FUNCTION_BLOCK IA_COGSOGRapidUpdate (* ISOBUS Adapter for Course Over Ground and Speed Over Ground (Rapid Update) *)
  (* Standard: NMEA 2000; Classification: PGN 129026; Description: Copyright (c) 2024-2026 HR Agrartechnik GmbH This program and the accompanying materials are made available under the terms of the Eclipse Public License 2.0 which is available at https://www.eclipse.org/legal/epl-2.0/ SPDX-License-Identifier: EPL-2.0 *)
  (* Version 1.4, 2026-09-17, Franz Höpfinger, HR Agrartechnik GmbH, Dokumentation (Franz: 'das passt, wir dokumentieren das in den Bausteinen. E_D_FF ist ein IEC 61499 Standardbaustein, wir halten uns STRENG an die Norm. E_D_FF_ANY ist davon abgeleitet, sollte sich gleich verhalten'): E_D_FF_Timeout (E_D_FF, IEC 61499-1 Annex A Standardbaustein) feuert EO NICHT beim allerersten CLK, wenn der erste echte Wert mit dem default-initialisierten Vergleichszustand (FALSE) uebereinstimmt - bleibt I_CORE.Q_timeout von Anfang an FALSE (Normalfall, kein Timeout), feuert TIMEOUT.E1 nie initial. Bewusst kein Bug, sondern standardkonformes Verhalten (analog E_RS/E_SR, wo genau dasselbe Verhalten Anlass fuer die Sonderformen E_RS_SYM/E_SR_SYM war) - hier bewusst KEINE eigene SYM-Variante, da nachgelagerte Verbraucher TIMEOUT.D1 als Datenwert lesen, nicht nur das Event. *)
  (* Version 1.3, 2026-09-17, Franz Höpfinger, HR Agrartechnik GmbH, Bugfix (PR #241 Review, qodo-code-review[bot]: 'Normal traffic floods timeout consumers - every IND republishes Q_timeout even when it did not change'): E_D_FF_Timeout (E_D_FF_ANY) vor TIMEOUT eingefuegt, wie schon fuer die anderen Signale dieser Datei - I_CORE.TIMEOUT und I_CORE.IND feuern jetzt beide nur noch E_D_FF_Timeout.CLK, TIMEOUT.E1/D1 werden nur noch bei tatsaechlicher Aenderung von Q_timeout aktualisiert, nicht mehr bei jeder einzelnen Botschaft im gesunden Normalbetrieb. *)
  (* Version 1.2, 2026-09-17, Franz Höpfinger, HR Agrartechnik GmbH, Bugfix (Franz: 'IA_VDS hat einen Bug, moeglicherweise alle anderen auch'): .IND->TIMEOUT.E1 ergaenzt (analog IA_VDS) - bisher wurde TIMEOUT.E1 NUR von .TIMEOUT gefeuert (Timeout-Beginn), nie beim Eintreffen einer normalen Botschaft (.IND) - TIMEOUT.D1 (Q_timeout=FALSE) wurde also gesetzt, aber nie an den TIMEOUT-Plug propagiert, sobald der Timeout wieder endete. *)
  (* Version 1.1, 2026-09-16, Franz Höpfinger, HR Agrartechnik GmbH, E_D_FF_ANY-Aenderungsfilter fuer COG/SOG/SID/COG_REF ergaenzt (analog IA_RPTO v1.1) - I_CORE.IND feuerte bisher bei jeder Botschaft unbedingt, auch ohne Wertaenderung. *)
  PACKAGE isobus::tecu;
  (* Documentation:
  ISOBUS Adapter for Course Over Ground and Speed Over Ground (Rapid Update)
   TIMEOUT.E1-Verdrahtung: I_CORE.TIMEOUT (echter Timeout-Eintritt) UND I_CORE.IND (Normalbetrieb) feuern beide E_D_FF_Timeout.CLK; E_D_FF_Timeout (E_D_FF_ANY, gespeist von I_CORE.Q_timeout) laesst TIMEOUT.E1 nur bei tatsaechlicher Wertaenderung durch - so wird TIMEOUT.D1 (Q_timeout) am Adapter-Plug beim Zuruecksetzen auf false weiterhin zuverlaessig aktualisiert, ohne bei jeder einzelnen Botschaft im gesunden Normalbetrieb erneut zu feuern. Der zugrundeliegende TIMEOUT/IND-Vertrag von I_CORE selbst ist in dessen eigener .fbt-Datei dokumentiert.
  *)
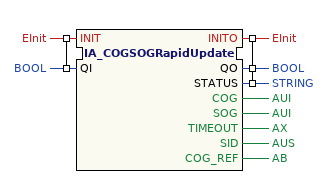
  EVENT_INPUT
    INIT : EInit WITH QI; (* Service Initialization *)
  END_EVENT
  EVENT_OUTPUT
    INITO : EInit WITH QO, STATUS; (* Initialization Confirm *)
  END_EVENT
  VAR_INPUT
    QI : BOOL; (* Event Input Qualifier *)
  END_VAR
  VAR_OUTPUT
    QO : BOOL; (* Event Output Qualifier *)
    STATUS : STRING;
  END_VAR
  PLUGS
    COG : adapter::types::unidirectional::AUI; (* Course Over Ground *)
    SOG : adapter::types::unidirectional::AUI; (* Speed Over Ground *)
    TIMEOUT : adapter::types::unidirectional::AX; (* Timeout Status *)
    SID : adapter::types::unidirectional::AUS; (* Sequence ID *)
    COG_REF : adapter::types::unidirectional::AB; (* COG Reference *)
  END_PLUGS
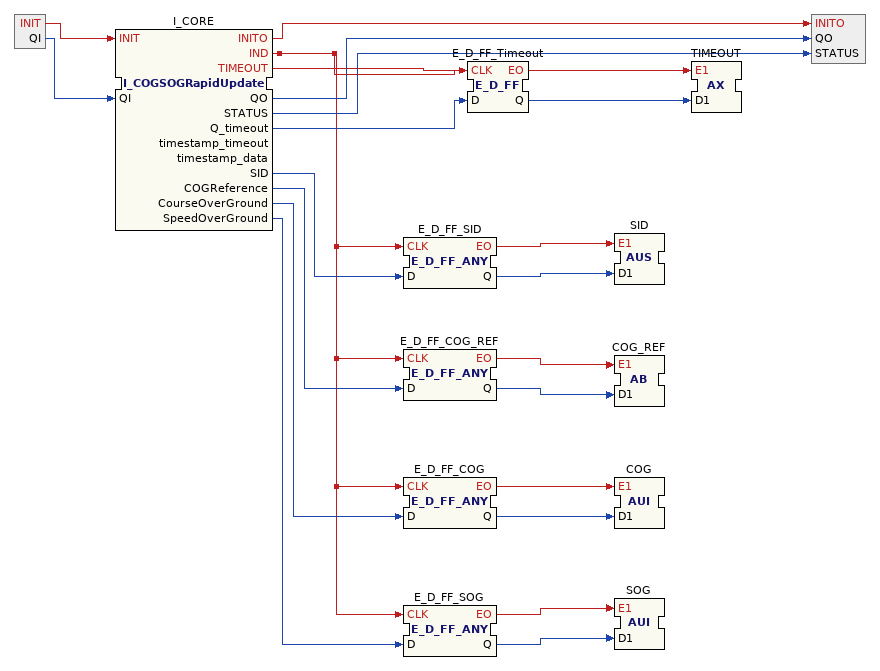
  FBS
    I_CORE : isobus::tecu::I_COGSOGRapidUpdate;
    E_D_FF_COG : iec61499::events::E_D_FF_ANY;
    E_D_FF_SOG : iec61499::events::E_D_FF_ANY;
    E_D_FF_SID : iec61499::events::E_D_FF_ANY;
    E_D_FF_COG_REF : iec61499::events::E_D_FF_ANY;
    E_D_FF_Timeout : iec61499::events::E_D_FF;
  END_FBS
  EVENT_CONNECTIONS
    INIT TO I_CORE.INIT;
    I_CORE.INITO TO INITO;
    I_CORE.IND TO E_D_FF_COG.CLK;
    E_D_FF_COG.EO TO COG.E1;
    I_CORE.IND TO E_D_FF_SOG.CLK;
    E_D_FF_SOG.EO TO SOG.E1;
    I_CORE.IND TO E_D_FF_SID.CLK;
    E_D_FF_SID.EO TO SID.E1;
    I_CORE.IND TO E_D_FF_COG_REF.CLK;
    E_D_FF_COG_REF.EO TO COG_REF.E1;
    I_CORE.TIMEOUT TO E_D_FF_Timeout.CLK;
    I_CORE.IND TO E_D_FF_Timeout.CLK;
    E_D_FF_Timeout.EO TO TIMEOUT.E1;
  END_CONNECTIONS
  DATA_CONNECTIONS
    QI TO I_CORE.QI;
    I_CORE.QO TO QO;
    I_CORE.STATUS TO STATUS;
    I_CORE.CourseOverGround TO E_D_FF_COG.D;
    E_D_FF_COG.Q TO COG.D1;
    I_CORE.SpeedOverGround TO E_D_FF_SOG.D;
    E_D_FF_SOG.Q TO SOG.D1;
    I_CORE.Q_timeout TO E_D_FF_Timeout.D;
    E_D_FF_Timeout.Q TO TIMEOUT.D1;
    I_CORE.SID TO E_D_FF_SID.D;
    E_D_FF_SID.Q TO SID.D1;
    I_CORE.COGReference TO E_D_FF_COG_REF.D;
    E_D_FF_COG_REF.Q TO COG_REF.D1;
  END_CONNECTIONS
END_FUNCTION_BLOCK
